(* IEC 61131-3 sources: WebSocket/, 5 files *)

(* ---- Types.typ ---- *)
TYPE
	WSHeader_typ : 	STRUCT
		fin : BOOL;
		rsv : USINT;
		opCode : USINT;
		mask : BOOL;
		maskingKey : ARRAY[0..3]OF USINT;
		frameLength : UDINT;
	END_STRUCT;
	WS_OpCode_enum :
		(
		WS_OPCODE_CONTINUATION := 0,
		WS_OPCODE_TEXT := 1,
		WS_OPCODE_BINARY := 2,
		WS_OPCODE_RESERVED_NON_CONTROL := 3,
		WS_OPCODE_CONNECTION_CLOSE := 8,
		WS_OPCODE_PING := 9,
		WS_OPCODE_PONG := 10,
		WS_OPCODE_RESERVED_CONTROL := 11
		);
	WS_ERR_enum :
		(
		WS_ERR_OK,
		WS_ERR_INVALID_INPUT := 5500,
		WS_ERR_NOT_IMPLEMENTED,
		WS_ERR_PAYLOAD_LENGTH,
		WS_ERR_MEM_ALLOC,
		WS_ERR_NO_LICENSE,
		WS_ERR_KEY_NOT_FOUND, (*5505*)
		WS_ERR_PARTIAL_HTTP_MESSAGE,
		WS_ERR_INVALID_HTTP_MESSAGE,
		WS_ERR_BUFFER_FULL,
		WS_ERR_ (*5509*)
		);
	WS_Mode_enum :
		(
		WS_MODE_SERVER := 50000,
		WS_MODE_CLIENT
		);
	MaskingKey_typ :ARRAY[0..3]OF USINT;
END_TYPE

(*Internal types*)

TYPE
	WSDecode_Internal_typ : 	STRUCT
		mask : wsMask;
	END_STRUCT;
	WSEncode_Internal_typ : 	STRUCT
		mask : wsMask;
	END_STRUCT;
	WSConnect_Internal_typ : 	STRUCT
		encodeBase64 : httpEncodeBase64;
	END_STRUCT;
END_TYPE

(* ---- WSMgr.typ ---- *)
TYPE
	WSConnectionManager_typ : 	STRUCT
		in : WSConnectionManager_In_typ;
		out : WSConnectionManager_Out_typ;
		internal : WSConnectionManager_Internal_typ;
	END_STRUCT;
	WSConnectionManager_In_typ : 	STRUCT
		cmd : WSConnectionManager_In_Cmd_typ;
		cfg : WSConnectionManager_In_Cfg_typ;
	END_STRUCT;
	WSConnectionManager_In_Cmd_typ : 	STRUCT
		enable : BOOL;
		acknowledgeConnection : BOOL;
		acknowledgeError : BOOL;
	END_STRUCT;
	WSConnectionManager_In_Cfg_typ : 	STRUCT
		mode : WS_Mode_enum;
		localIPAddress : STRING[TCPCOMM_STRLEN_IPADDRESS];
		localPort : UDINT;
		remoteIPAddress : STRING[TCPCOMM_STRLEN_IPADDRESS];
		remotePort : UDINT;
		sendBufferSize : UDINT;
		useSSL : BOOL;
		sslCertificate : UDINT;
	END_STRUCT;
	WSConnectionManager_Out_typ : 	STRUCT
		newConnectionAvailable : BOOL;
		connection : WSConnectionManager_Desc_typ;
		error : BOOL;
		errorID : UINT;
		errorString : STRING[WS_STRLEN_ERRORSTRING];
	END_STRUCT;
	WSConnectionManager_Desc_typ : 	STRUCT
		parameters : TCPConnection_Desc_typ;
		mode : WS_Mode_enum;
	END_STRUCT;
	WSConnectionManager_Internal_typ : 	STRUCT
		tcpConnection : TCPConnectionMgr_typ;
	END_STRUCT;
END_TYPE

(* ---- WSStream.typ ---- *)
(*For each client lets instantiate an interface*)

TYPE
	WSStream_typ : 	STRUCT
		in : WSStream_IN_typ;
		out : WSStream_OUT_typ;
		internal : WSStream_Internal_typ;
	END_STRUCT;
	WSStream_IN_typ : 	STRUCT
		cmd : WSStream_IN_CMD_typ;
		par : WSStream_IN_PAR_typ;
		cfg : WSStream_IN_CFG_typ;
	END_STRUCT;
	WSStream_IN_CMD_typ : 	STRUCT
		receive : BOOL;
		send : BOOL;
		close : BOOL;
		acknowledgeData : BOOL;
		acknowledgeError : BOOL;
	END_STRUCT;
	WSStream_IN_PAR_typ : 	STRUCT
		connection : WSConnectionManager_Desc_typ;
		pReceiveData : UDINT;
		maxReceiveLength : UDINT;
		receiveFlags : UINT;
		allowContinuousReceive : BOOL;
		pSendData : UDINT;
		sendLength : UDINT;
		sendHeader : WSHeader_typ;
		sendFlags : UINT;
		allowContinuousSend : BOOL;
	END_STRUCT;
	WSStream_IN_CFG_typ : 	STRUCT
		bufferSize : UDINT;
	END_STRUCT;
	WSStream_OUT_typ : 	STRUCT
		connection : WSConnectionManager_Desc_typ;
		active : BOOL;
		connected : BOOL;
		receiving : BOOL;
		header : WSHeader_typ;
		partialDataReceived : BOOL;
		dataReceived : BOOL;
		receivedDataLength : UDINT;
		sending : BOOL;
		dataSent : BOOL;
		sentDataLength : UDINT;
		error : BOOL;
		errorID : UINT;
		errorString : STRING[TCPCOMM_STRLEN_ERRORSTRING];
	END_STRUCT;
	WSStream_Internal_typ : 	STRUCT
		debug : WSStream_Int_Debug_typ;
		fub : WSStream_Int_FUB_typ;
		connection : WSConnectionManager_Desc_typ;
		initialized : BOOL;
		connected : BOOL;
		connectionUpgraded : BOOL;
		connectionState : UINT;
		bufferSize : UDINT;
		sendBuffer : UDINT;
		recieveBuffer : UDINT;
		prevSend : BOOL;
	END_STRUCT;
	WSStream_Int_Debug_typ : 	STRUCT
		New_Member : USINT;
	END_STRUCT;
	WSStream_Int_FUB_typ : 	STRUCT
		tcpStream : TCPStream_typ;
		wsDecode : wsDecode;
		wsEncode : wsEncode;
		wsConnect : wsConnect;
		wsMask : wsMask;
	END_STRUCT;
END_TYPE

(* ---- WebSocket.fun ---- *)
(*Main Fns*)

FUNCTION wsManageConnection : BOOL
	VAR_INPUT
		inst : WSConnectionManager_typ;
	END_VAR
END_FUNCTION

FUNCTION wsSend : BOOL
	VAR_INPUT
		inst : WSStream_typ;
	END_VAR
END_FUNCTION

FUNCTION wsReceive : BOOL
	VAR_INPUT
		inst : WSStream_typ;
	END_VAR
END_FUNCTION
(*Utility Fns*)

FUNCTION wsGetErrorMsg : UDINT
	VAR_INPUT
		dest : UDINT;
		errorID : DINT;
		destSize : UDINT;
	END_VAR
END_FUNCTION

FUNCTION wsModeIsValid : BOOL
	VAR_INPUT
		mode : DINT;
	END_VAR
END_FUNCTION
(*Low Level Fns*)

FUNCTION_BLOCK wsConnect (*Negotiate a new WebSocket connection TODO: Figure out how to add functionality later*) (*$GROUP=User,$CAT=User,$GROUPICON=User.png,$CATICON=User.png*)
	VAR_INPUT
		pInputMessage : UDINT;
		pOutputMessage : UDINT;
		outputMessageSize : UDINT;
	END_VAR
	VAR_OUTPUT
		status : UINT;
		outputMessageLength : UDINT;
	END_VAR
	VAR
		internal : WSConnect_Internal_typ;
	END_VAR
END_FUNCTION_BLOCK

FUNCTION_BLOCK wsDecode (*Decode a WebSocket frame*) (*$GROUP=User,$CAT=User,$GROUPICON=User.png,$CATICON=User.png*)
	VAR_INPUT
		pFrame : UDINT;
		frameLength : UDINT;
		pPayload : UDINT;
		payloadSize : UDINT;
	END_VAR
	VAR_OUTPUT
		status : UINT;
		partialHeader : BOOL;
		partialFrame : BOOL;
		fin : BOOL;
		rsv : USINT;
		opCode : USINT;
		mask : BOOL;
		maskingKey : MaskingKey_typ;
		headerLength : UDINT;
		payloadLength : UDINT;
		decodeLength : UDINT;
	END_VAR
	VAR
		internal : WSDecode_Internal_typ;
	END_VAR
END_FUNCTION_BLOCK

FUNCTION_BLOCK wsEncode (*Encode data into a WebSocket frame*) (*$GROUP=User,$CAT=User,$GROUPICON=User.png,$CATICON=User.png*)
	VAR_INPUT
		pFrame : UDINT;
		frameSize : UDINT;
		fin : BOOL;
		rsv : USINT;
		opCode : USINT;
		mask : BOOL; (*NOT SUPPORTED*)
		maskingKey : MaskingKey_typ; (*NOT SUPPORTED*)
		pPayload : UDINT;
		payloadLength : UDINT;
	END_VAR
	VAR_OUTPUT
		status : UINT;
		frameLength : UDINT;
	END_VAR
	VAR
		internal : WSEncode_Internal_typ;
	END_VAR
END_FUNCTION_BLOCK

FUNCTION_BLOCK wsMask (*Mask / Unmask Src into Dest*)
	VAR_INPUT
		src : UDINT; (*Pointer to STRING with original data*)
		srcLength : UDINT; (*Length of data*)
		dest : UDINT; (*Pointer to STRING to destination*)
		destSize : UDINT; (*Size of destination*)
		maskingKey : MaskingKey_typ; (*Masking Key, if 0 then a key will be generated*)
	END_VAR
	VAR_OUTPUT
		status : UINT;
		destLength : UDINT; (*Length of dest*)
	END_VAR
END_FUNCTION_BLOCK

(* ---- Constants.var ---- *)
VAR CONSTANT
	WS_HEADER_MAX_LEN : USINT := 14;
	WS_HEADER_MIN_LEN : USINT := 2;
	WS_STRLEN_ERRORSTRING : UINT := 320;
	WS_STRLEN_CONNECTMESSAGE : USINT := 129;
	WS_STRLEN_KEYHEADER : UINT := 18;
	WS_SOC_MAGICSTRING : STRING[36] := '258EAFA5-E914-47DA-95CA-C5AB0DC85B11';
	WS_DEFAULT_CONNECT_BUF_SIZE : UINT := 1000;
END_VAR
